(* PLC project Test.project, CODESYS CODESYS V3.5 SP21 Patch 5 *)
(* stored: creationDateTime 2026-05-07T14:55:41.6791703, modificationDateTime 2026-05-07T14:54:46.6861198 *)

PROGRAM PLC_PRG
  VAR
    counter : INT;
  END_VAR

                    counter := counter + 1;

IF counter > 100 THEN
	counter := 0;
END_IF
                  
END_PROGRAM

CONFIGURATION Device
  RESOURCE Application ON PLC
    TASK MainTask(INTERVAL := T#50ms, PRIORITY := 15);
    PROGRAM PLC_PRG WITH MainTask : PLC_PRG;
  END_RESOURCE
END_CONFIGURATION

CONFIGURATION Kbus
END_CONFIGURATION

CONFIGURATION Serial
END_CONFIGURATION

CONFIGURATION COM1
END_CONFIGURATION
